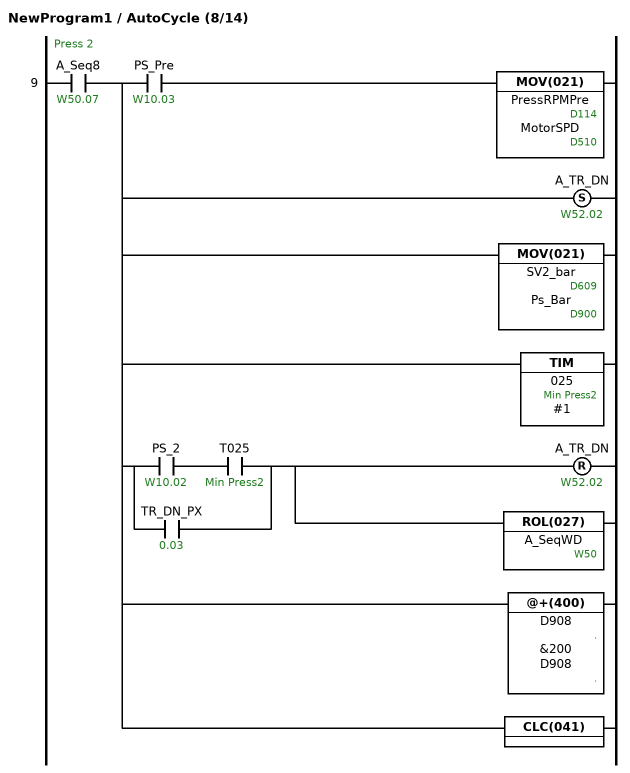
; [picture p24: NewProgram1 / AutoCycle, rungs 9-9]
; rung 9: Press 2
LD A_Seq8  ; W50.07
OUT TR0
AND PS_Pre  ; W10.03
MOV(021) PressRPMPre MotorSPD  ; D114, D510
LD TR0
SET A_TR_DN  ; W52.02
MOV(021) SV2_bar Ps_Bar  ; D609, D900
TIM 025 #1  ; Min Press2
LD PS_2  ; W10.02
AND T025  ; Min Press2
OR TR_DN_PX  ; 0.03
ANDLD
RSET A_TR_DN  ; W52.02
ROL(027) A_SeqWD  ; W50
LD TR0
@+(400) D908 &200 D908  ; .
CLC(041)

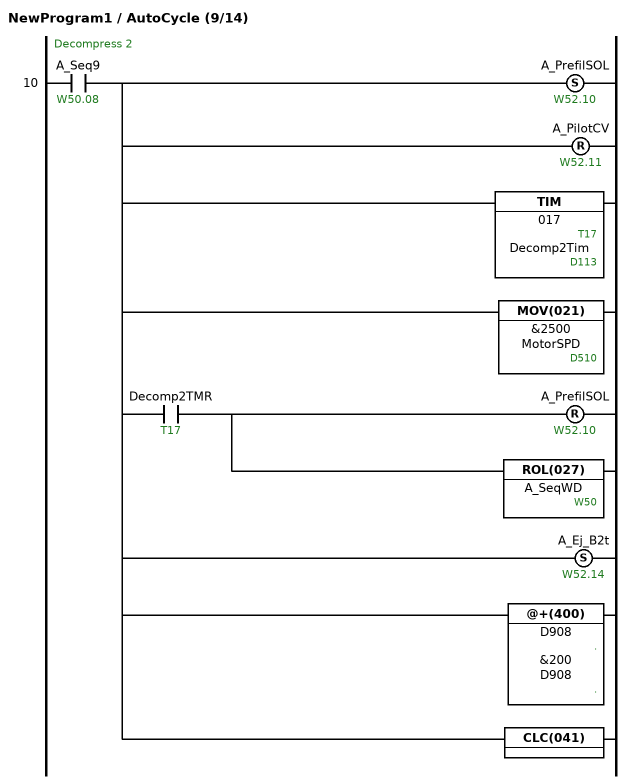
; rung 10: Decompress 2
LD A_Seq9  ; W50.08
OUT TR0
SET A_PrefilSOL  ; W52.10
RSET A_PilotCV  ; W52.11
TIM 017 Decomp2Tim  ; D113, T17
MOV(021) &2500 MotorSPD  ; D510
AND Decomp2TMR  ; T17
RSET A_PrefilSOL  ; W52.10
ROL(027) A_SeqWD  ; W50
LD TR0
SET A_Ej_B2t  ; W52.14
@+(400) D908 &200 D908  ; .
CLC(041)

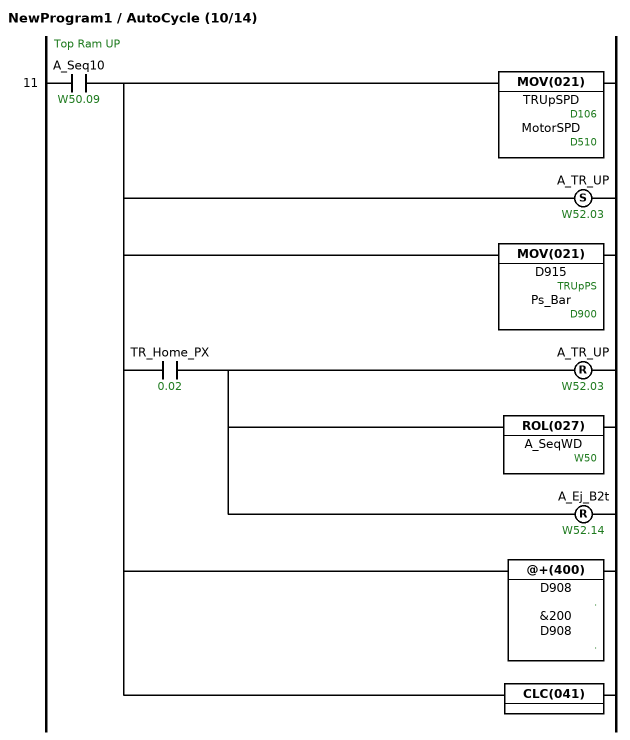
; rung 11: Top Ram UP
LD A_Seq10  ; W50.09
OUT TR0
MOV(021) TRUpSPD MotorSPD  ; D106, D510
SET A_TR_UP  ; W52.03
MOV(021) D915 Ps_Bar  ; TRUpPS, D900
AND TR_Home_PX  ; 0.02
RSET A_TR_UP  ; W52.03
ROL(027) A_SeqWD  ; W50
RSET A_Ej_B2t  ; W52.14
LD TR0
@+(400) D908 &200 D908  ; .
CLC(041)

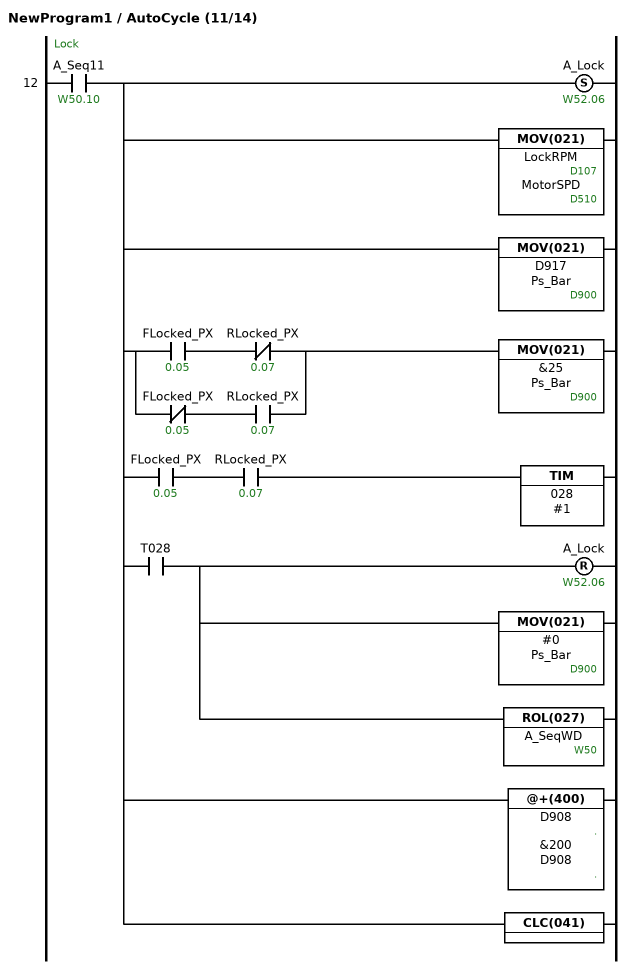
; rung 12: Lock
LD A_Seq11  ; W50.10
OUT TR0
SET A_Lock  ; W52.06
MOV(021) LockRPM MotorSPD  ; D107, D510
MOV(021) D917 Ps_Bar  ; D900
LD FLocked_PX  ; 0.05
ANDNOT RLocked_PX  ; 0.07
LDNOT FLocked_PX  ; 0.05
AND RLocked_PX  ; 0.07
ORLD
ANDLD
MOV(021) &25 Ps_Bar  ; D900
LD TR0
AND FLocked_PX  ; 0.05
AND RLocked_PX  ; 0.07
TIM 028 #1
LD TR0
AND T028
RSET A_Lock  ; W52.06
MOV(021) #0 Ps_Bar  ; D900
ROL(027) A_SeqWD  ; W50
LD TR0
@+(400) D908 &200 D908  ; .
CLC(041)

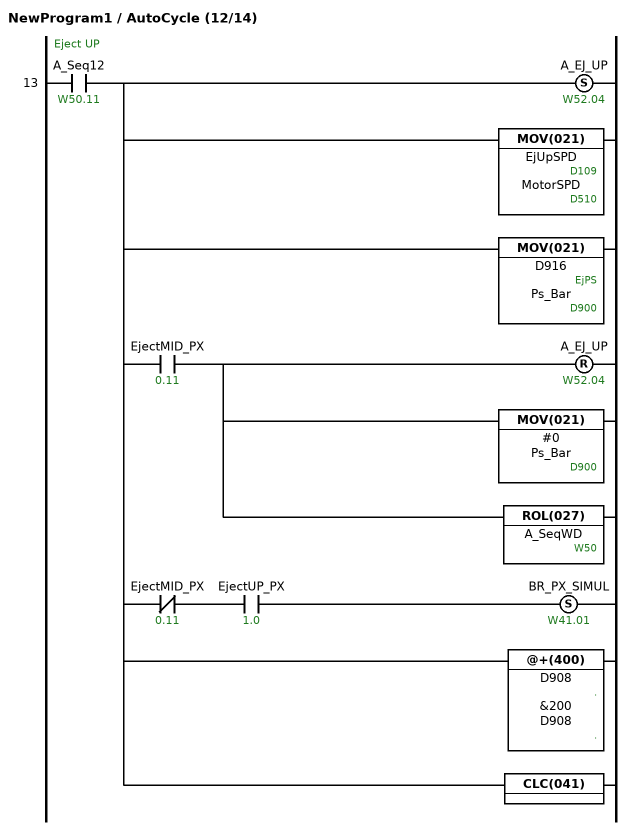
; rung 13: Eject UP
LD A_Seq12  ; W50.11
OUT TR0
SET A_EJ_UP  ; W52.04
MOV(021) EjUpSPD MotorSPD  ; D109, D510
MOV(021) D916 Ps_Bar  ; EjPS, D900
AND EjectMID_PX  ; 0.11
RSET A_EJ_UP  ; W52.04
MOV(021) #0 Ps_Bar  ; D900
ROL(027) A_SeqWD  ; W50
LD TR0
ANDNOT EjectMID_PX  ; 0.11
AND EjectUP_PX  ; 1.0
SET BR_PX_SIMUL  ; W41.01
LD TR0
@+(400) D908 &200 D908  ; .
CLC(041)

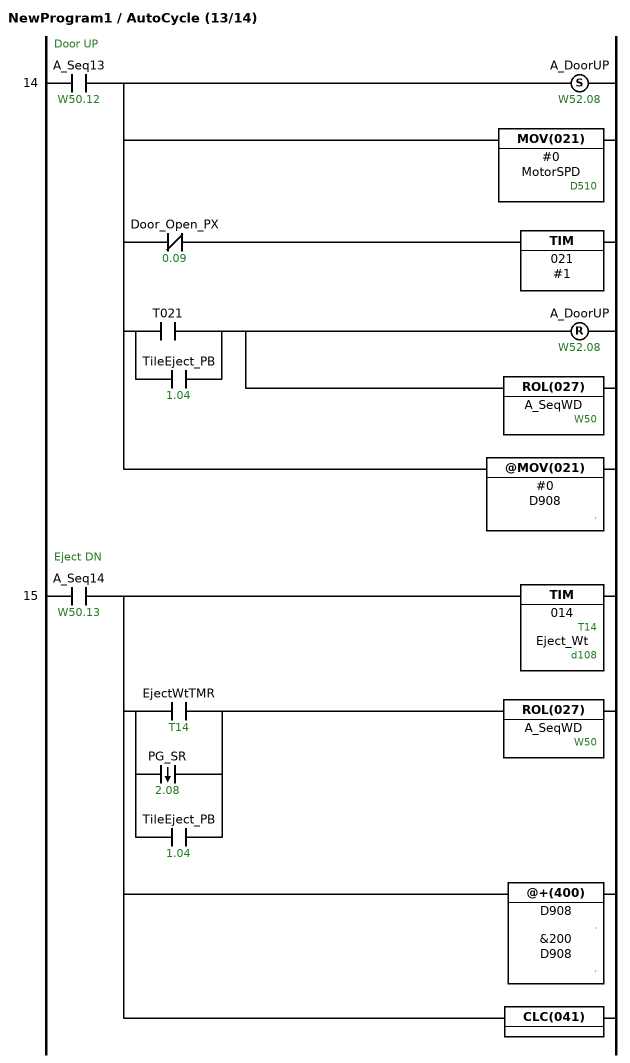
; rung 14: Door UP
LD A_Seq13  ; W50.12
OUT TR0
SET A_DoorUP  ; W52.08
MOV(021) #0 MotorSPD  ; D510
ANDNOT Door_Open_PX  ; 0.09
TIM 021 #1
LD TR0
LD T021
OR TileEject_PB  ; 1.04
ANDLD
RSET A_DoorUP  ; W52.08
ROL(027) A_SeqWD  ; W50
LD TR0
@MOV(021) #0 D908  ; .
; rung 15: Eject DN
LD A_Seq14  ; W50.13
OUT TR0
TIM 014 Eject_Wt  ; d108, T14
LD EjectWtTMR  ; T14
%OR PG_SR  ; 2.08
OR TileEject_PB  ; 1.04
ANDLD
ROL(027) A_SeqWD  ; W50
LD TR0
@+(400) D908 &200 D908  ; .
CLC(041)

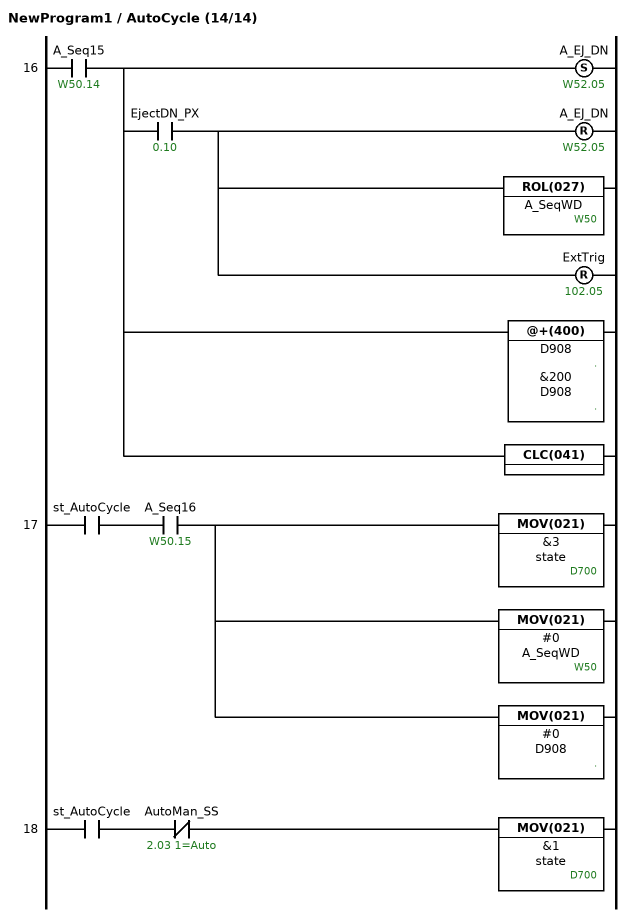
; rung 16
LD A_Seq15  ; W50.14
OUT TR0
SET A_EJ_DN  ; W52.05
AND EjectDN_PX  ; 0.10
RSET A_EJ_DN  ; W52.05
ROL(027) A_SeqWD  ; W50
RSET ExtTrig  ; 102.05
LD TR0
@+(400) D908 &200 D908  ; .
CLC(041)
; rung 17
LD st_AutoCycle
AND A_Seq16  ; W50.15
MOV(021) &3 state  ; D700
MOV(021) #0 A_SeqWD  ; W50
MOV(021) #0 D908  ; .
; rung 18
LD st_AutoCycle
ANDNOT AutoMan_SS  ; 2.03 1=Auto
MOV(021) &1 state  ; D700

### Section AutoReq

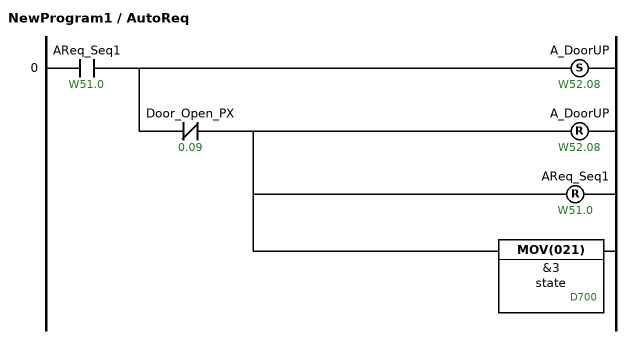
; rung 0
LD AReq_Seq1  ; W51.0
SET A_DoorUP  ; W52.08
ANDNOT Door_Open_PX  ; 0.09
RSET A_DoorUP  ; W52.08
RSET AReq_Seq1  ; W51.0
MOV(021) &3 state  ; D700

### Section TileEject

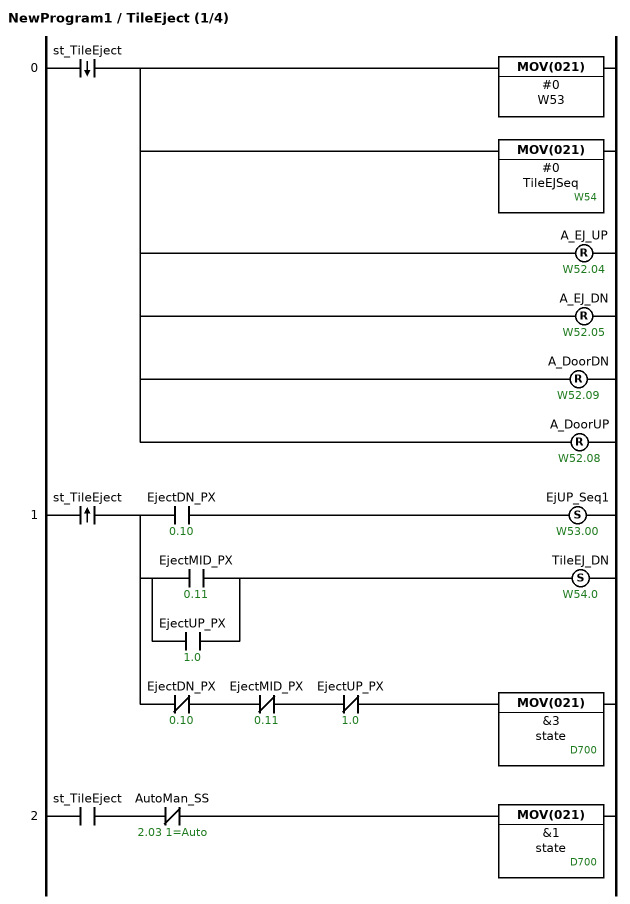
; rung 0
%LD st_TileEject
MOV(021) #0 W53
MOV(021) #0 TileEJSeq  ; W54
RSET A_EJ_UP  ; W52.04
RSET A_EJ_DN  ; W52.05
RSET A_DoorDN  ; W52.09
RSET A_DoorUP  ; W52.08
; rung 1
@LD st_TileEject
OUT TR0
AND EjectDN_PX  ; 0.10
SET EjUP_Seq1  ; W53.00
LD TR0
LD EjectMID_PX  ; 0.11
OR EjectUP_PX  ; 1.0
ANDLD
SET TileEJ_DN  ; W54.0
LD TR0
ANDNOT EjectDN_PX  ; 0.10
ANDNOT EjectMID_PX  ; 0.11
ANDNOT EjectUP_PX  ; 1.0
MOV(021) &3 state  ; D700
; rung 2
LD st_TileEject
ANDNOT AutoMan_SS  ; 2.03 1=Auto
MOV(021) &1 state  ; D700

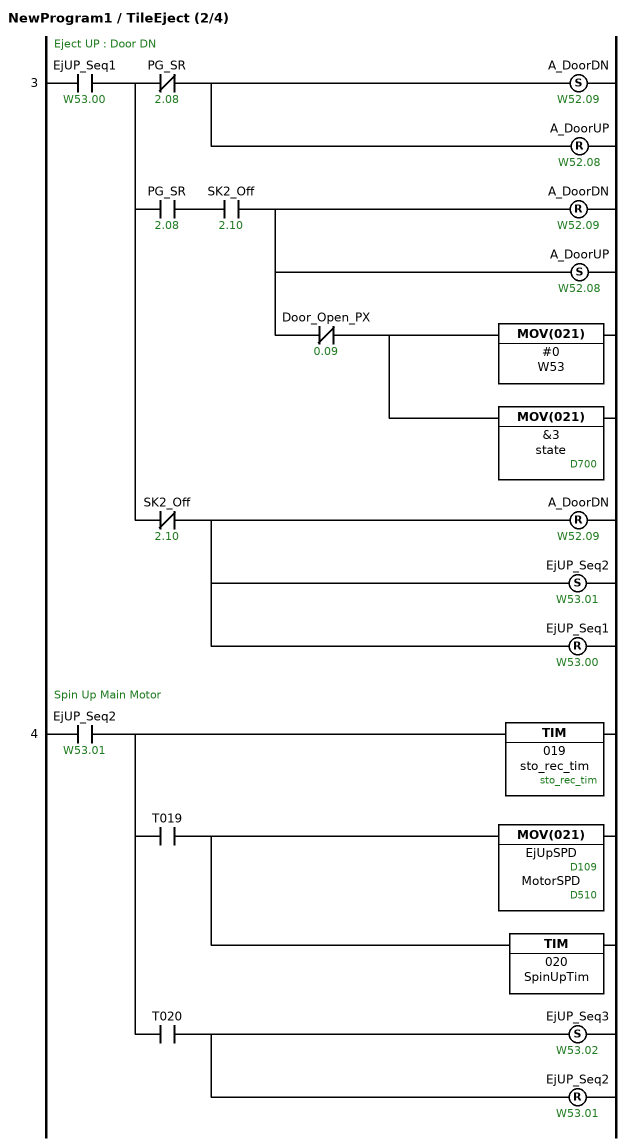
; rung 3: Eject UP : Door DN
LD EjUP_Seq1  ; W53.00
OUT TR0
ANDNOT PG_SR  ; 2.08
SET A_DoorDN  ; W52.09
RSET A_DoorUP  ; W52.08
LD TR0
AND PG_SR  ; 2.08
AND SK2_Off  ; 2.10
RSET A_DoorDN  ; W52.09
SET A_DoorUP  ; W52.08
ANDNOT Door_Open_PX  ; 0.09
MOV(021) #0 W53
MOV(021) &3 state  ; D700
LD TR0
ANDNOT SK2_Off  ; 2.10
RSET A_DoorDN  ; W52.09
SET EjUP_Seq2  ; W53.01
RSET EjUP_Seq1  ; W53.00
; rung 4: Spin Up Main Motor
LD EjUP_Seq2  ; W53.01
OUT TR0
TIM 019 sto_rec_tim  ; sto_rec_tim
AND T019
MOV(021) EjUpSPD MotorSPD  ; D109, D510
TIM 020 SpinUpTim
LD TR0
AND T020
SET EjUP_Seq3  ; W53.02
RSET EjUP_Seq2  ; W53.01

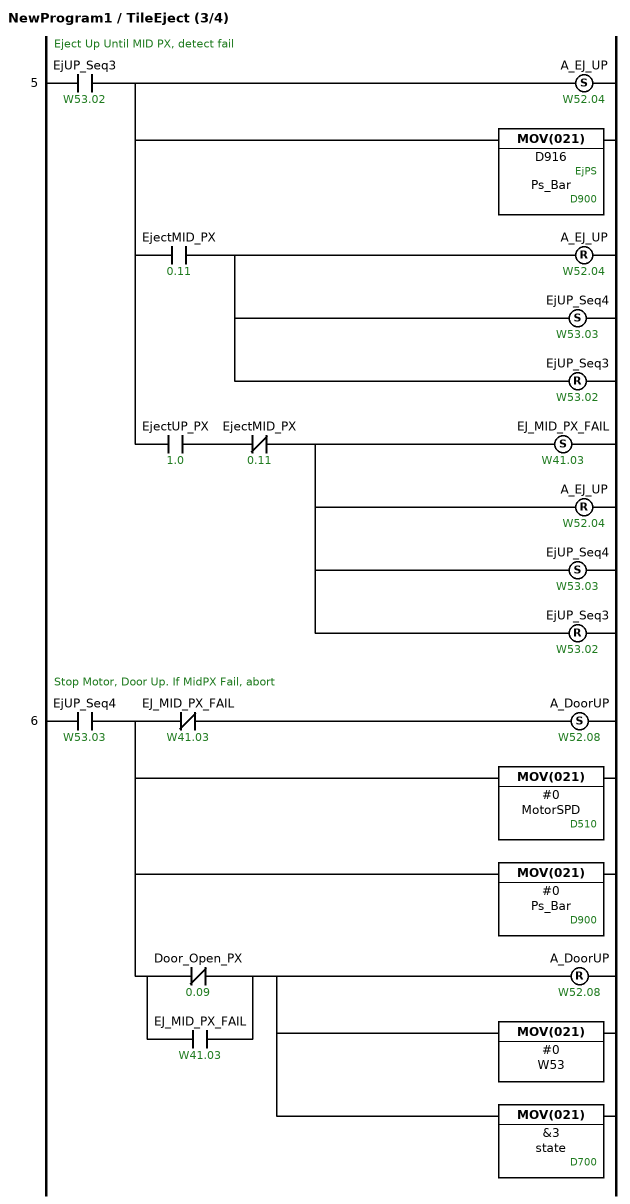
; rung 5: Eject Up Until MID PX, detect fail
LD EjUP_Seq3  ; W53.02
OUT TR0
SET A_EJ_UP  ; W52.04
MOV(021) D916 Ps_Bar  ; EjPS, D900
AND EjectMID_PX  ; 0.11
RSET A_EJ_UP  ; W52.04
SET EjUP_Seq4  ; W53.03
RSET EjUP_Seq3  ; W53.02
LD TR0
AND EjectUP_PX  ; 1.0
ANDNOT EjectMID_PX  ; 0.11
SET EJ_MID_PX_FAIL  ; W41.03
RSET A_EJ_UP  ; W52.04
SET EjUP_Seq4  ; W53.03
RSET EjUP_Seq3  ; W53.02
; rung 6: Stop Motor, Door Up. If MidPX Fail, abort
LD EjUP_Seq4  ; W53.03
OUT TR0
ANDNOT EJ_MID_PX_FAIL  ; W41.03
SET A_DoorUP  ; W52.08
LD TR0
MOV(021) #0 MotorSPD  ; D510
MOV(021) #0 Ps_Bar  ; D900
LDNOT Door_Open_PX  ; 0.09
OR EJ_MID_PX_FAIL  ; W41.03
ANDLD
RSET A_DoorUP  ; W52.08
MOV(021) #0 W53
MOV(021) &3 state  ; D700

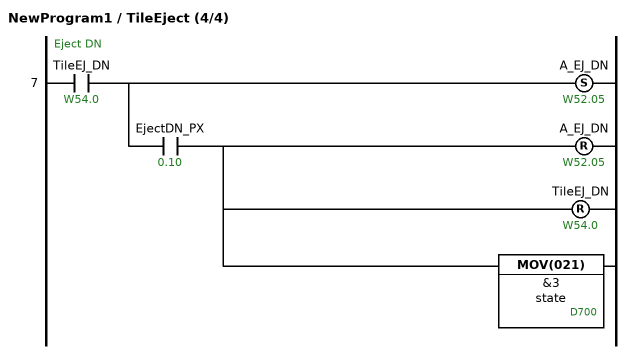
; rung 7: Eject DN
LD TileEJ_DN  ; W54.0
SET A_EJ_DN  ; W52.05
AND EjectDN_PX  ; 0.10
RSET A_EJ_DN  ; W52.05
RSET TileEJ_DN  ; W54.0
MOV(021) &3 state  ; D700

### Section MainMotorCtrl
; rung 0: 14.57 -> 3000, 14.59-> 3000

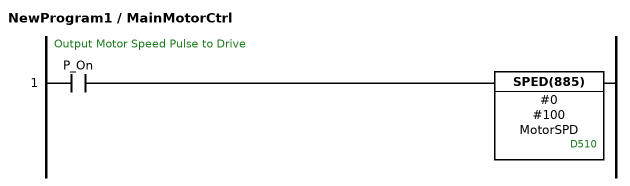
; rung 1: Output Motor Speed Pulse to Drive
LD P_On
SPED(885) #0 #100 MotorSPD  ; D510

### Section Outputs

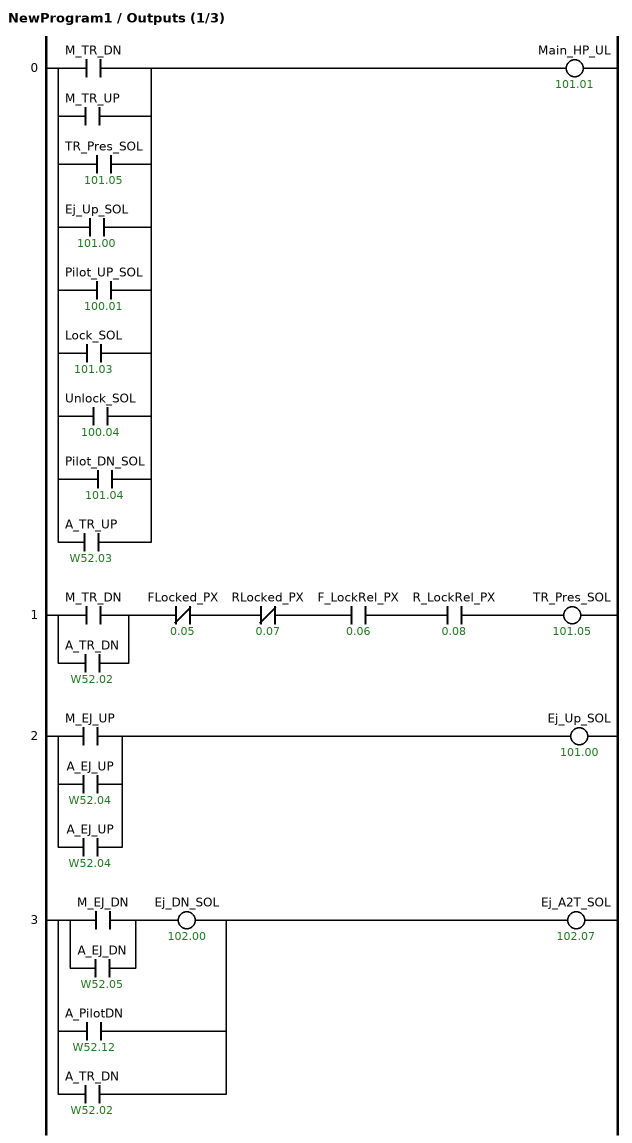
; rung 0
LD M_TR_DN
OR M_TR_UP
OR TR_Pres_SOL  ; 101.05
OR Ej_Up_SOL  ; 101.00
OR Pilot_UP_SOL  ; 100.01
OR Lock_SOL  ; 101.03
OR Unlock_SOL  ; 100.04
OR Pilot_DN_SOL  ; 101.04
OR A_TR_UP  ; W52.03
OUT Main_HP_UL  ; 101.01
; rung 1
LD M_TR_DN
OR A_TR_DN  ; W52.02
ANDNOT FLocked_PX  ; 0.05
ANDNOT RLocked_PX  ; 0.07
AND F_LockRel_PX  ; 0.06
AND R_LockRel_PX  ; 0.08
OUT TR_Pres_SOL  ; 101.05
; rung 2
LD M_EJ_UP
OR A_EJ_UP  ; W52.04
OR A_EJ_UP  ; W52.04
OUT Ej_Up_SOL  ; 101.00
; rung 3
LD M_EJ_DN
OR A_EJ_DN  ; W52.05
OUT Ej_DN_SOL  ; 102.00
LD A_PilotDN  ; W52.12
OR A_TR_DN  ; W52.02
ORLD
OUT Ej_A2T_SOL  ; 102.07

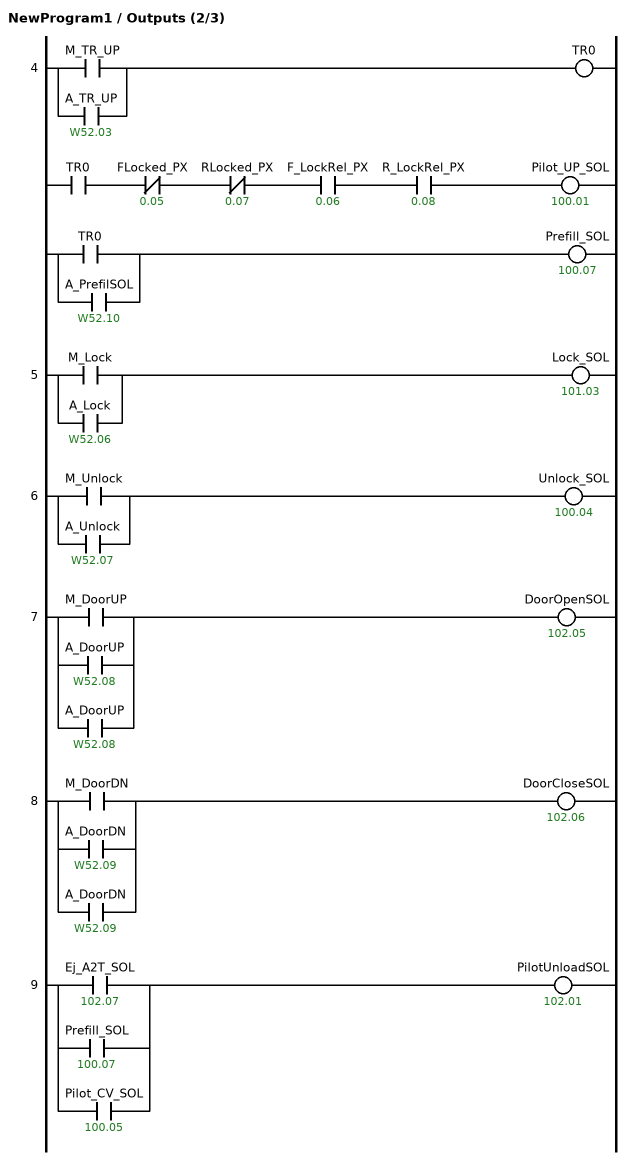
; rung 4
LD M_TR_UP
OR A_TR_UP  ; W52.03
OUT TR0
ANDNOT FLocked_PX  ; 0.05
ANDNOT RLocked_PX  ; 0.07
AND F_LockRel_PX  ; 0.06
AND R_LockRel_PX  ; 0.08
OUT Pilot_UP_SOL  ; 100.01
LD TR0
OR A_PrefilSOL  ; W52.10
OUT Prefill_SOL  ; 100.07
; rung 5
LD M_Lock
OR A_Lock  ; W52.06
OUT Lock_SOL  ; 101.03
; rung 6
LD M_Unlock
OR A_Unlock  ; W52.07
OUT Unlock_SOL  ; 100.04
; rung 7
LD M_DoorUP
OR A_DoorUP  ; W52.08
OR A_DoorUP  ; W52.08
OUT DoorOpenSOL  ; 102.05
; rung 8
LD M_DoorDN
OR A_DoorDN  ; W52.09
OR A_DoorDN  ; W52.09
OUT DoorCloseSOL  ; 102.06
; rung 9
LD Ej_A2T_SOL  ; 102.07
OR Prefill_SOL  ; 100.07
OR Pilot_CV_SOL  ; 100.05
OUT PilotUnloadSOL  ; 102.01

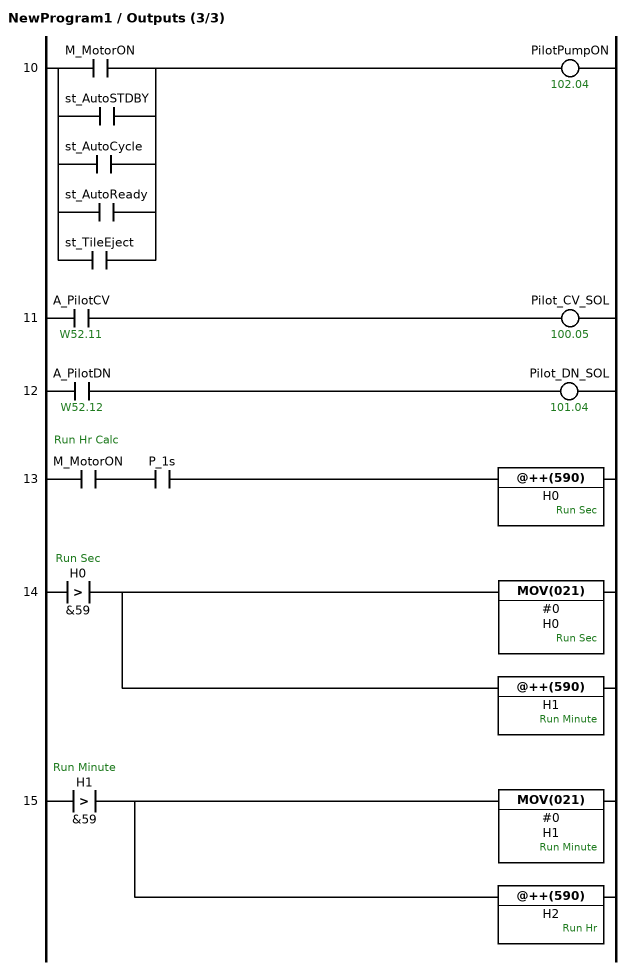
; rung 10
LD M_MotorON
OR st_AutoSTDBY
OR st_AutoCycle
OR st_AutoReady
OR st_TileEject
OUT PilotPumpON  ; 102.04
; rung 11
LD A_PilotCV  ; W52.11
OUT Pilot_CV_SOL  ; 100.05
; rung 12
LD A_PilotDN  ; W52.12
OUT Pilot_DN_SOL  ; 101.04
; rung 13: Run Hr Calc
LD M_MotorON
AND P_1s
@++(590) H0  ; Run Sec
; rung 14
LD>(320) H0 &59  ; Run Sec
MOV(021) #0 H0  ; Run Sec
@++(590) H1  ; Run Minute
; rung 15
LD>(320) H1 &59  ; Run Minute
MOV(021) #0 H1  ; Run Minute
@++(590) H2  ; Run Hr

### Section Profile

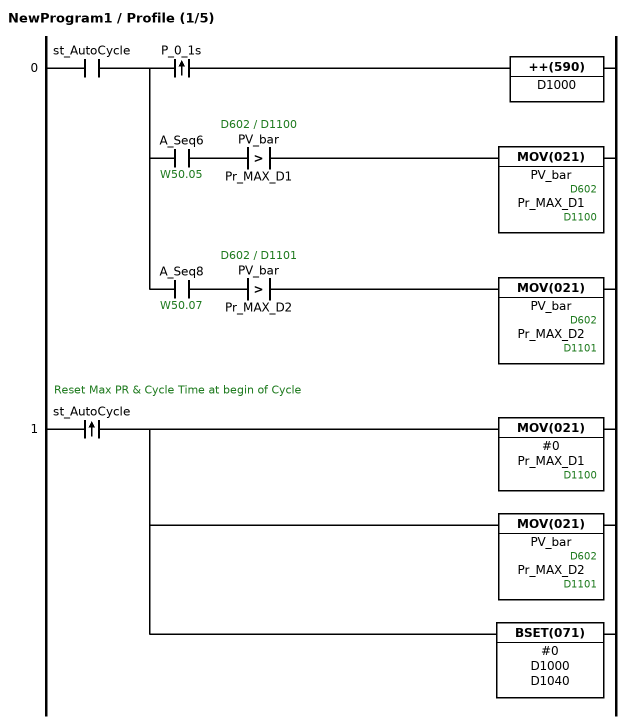
; rung 0
LD st_AutoCycle
OUT TR0
@AND P_0_1s
++(590) D1000
LD TR0
AND A_Seq6  ; W50.05
AND>(320) PV_bar Pr_MAX_D1  ; D602, D1100
MOV(021) PV_bar Pr_MAX_D1  ; D602, D1100
LD TR0
AND A_Seq8  ; W50.07
AND>(320) PV_bar Pr_MAX_D2  ; D602, D1101
MOV(021) PV_bar Pr_MAX_D2  ; D602, D1101
; rung 1: Reset Max PR & Cycle Time at begin of Cycle
@LD st_AutoCycle
MOV(021) #0 Pr_MAX_D1  ; D1100
MOV(021) PV_bar Pr_MAX_D2  ; D602, D1101
BSET(071) #0 D1000 D1040

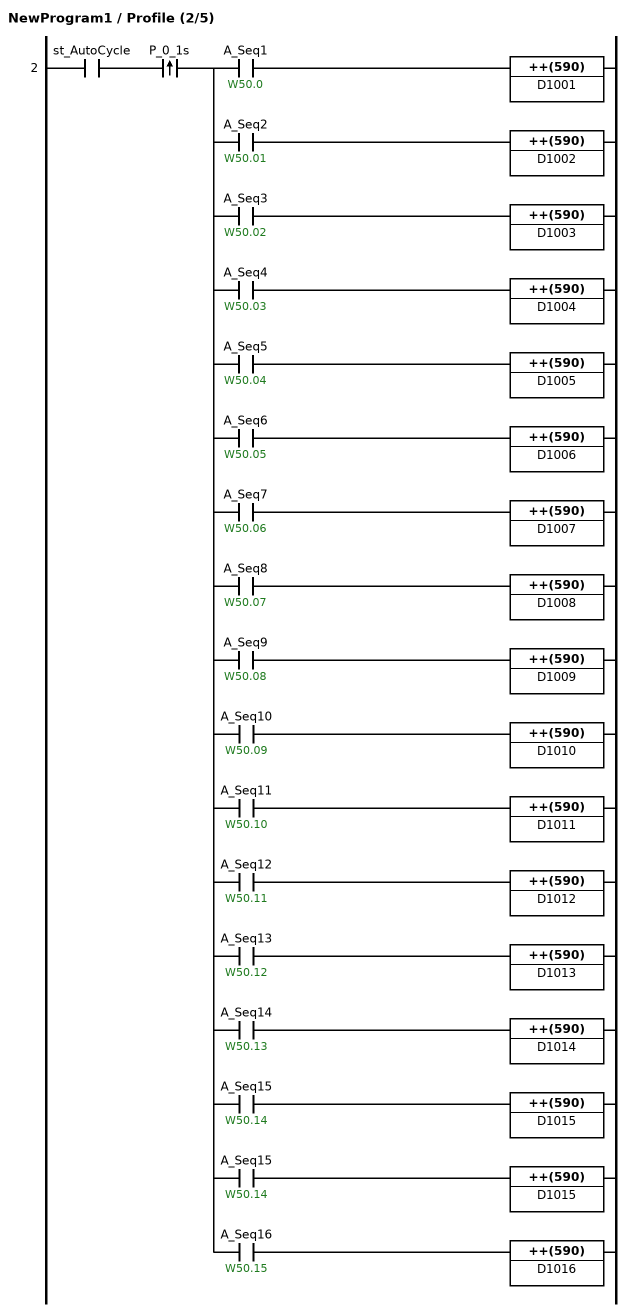
; rung 2
LD st_AutoCycle
@AND P_0_1s
OUT TR0
AND A_Seq1  ; W50.0
++(590) D1001
LD TR0
AND A_Seq2  ; W50.01
++(590) D1002
LD TR0
AND A_Seq3  ; W50.02
++(590) D1003
LD TR0
AND A_Seq4  ; W50.03
++(590) D1004
LD TR0
AND A_Seq5  ; W50.04
++(590) D1005
LD TR0
AND A_Seq6  ; W50.05
++(590) D1006
LD TR0
AND A_Seq7  ; W50.06
++(590) D1007
LD TR0
AND A_Seq8  ; W50.07
++(590) D1008
LD TR0
AND A_Seq9  ; W50.08
++(590) D1009
LD TR0
AND A_Seq10  ; W50.09
++(590) D1010
LD TR0
AND A_Seq11  ; W50.10
++(590) D1011
LD TR0
AND A_Seq12  ; W50.11
++(590) D1012
LD TR0
AND A_Seq13  ; W50.12
++(590) D1013
LD TR0
AND A_Seq14  ; W50.13
++(590) D1014
LD TR0
AND A_Seq15  ; W50.14
++(590) D1015
LD TR0
AND A_Seq15  ; W50.14
++(590) D1015
LD TR0
AND A_Seq16  ; W50.15
++(590) D1016

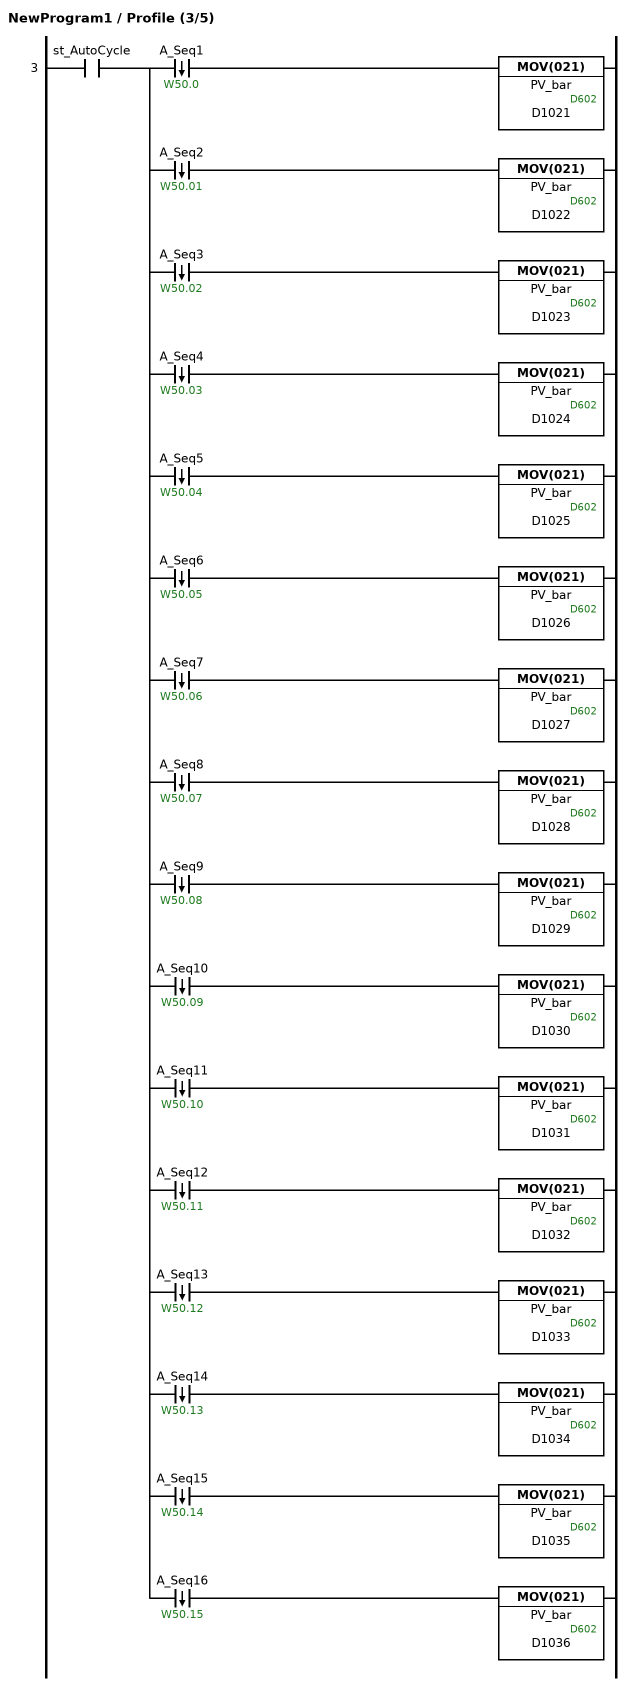
; rung 3
LD st_AutoCycle
OUT TR0
%AND A_Seq1  ; W50.0
MOV(021) PV_bar D1021  ; D602
LD TR0
%AND A_Seq2  ; W50.01
MOV(021) PV_bar D1022  ; D602
LD TR0
%AND A_Seq3  ; W50.02
MOV(021) PV_bar D1023  ; D602
LD TR0
%AND A_Seq4  ; W50.03
MOV(021) PV_bar D1024  ; D602
LD TR0
%AND A_Seq5  ; W50.04
MOV(021) PV_bar D1025  ; D602
LD TR0
%AND A_Seq6  ; W50.05
MOV(021) PV_bar D1026  ; D602
LD TR0
%AND A_Seq7  ; W50.06
MOV(021) PV_bar D1027  ; D602
LD TR0
%AND A_Seq8  ; W50.07
MOV(021) PV_bar D1028  ; D602
LD TR0
%AND A_Seq9  ; W50.08
MOV(021) PV_bar D1029  ; D602
LD TR0
%AND A_Seq10  ; W50.09
MOV(021) PV_bar D1030  ; D602
LD TR0
%AND A_Seq11  ; W50.10
MOV(021) PV_bar D1031  ; D602
LD TR0
%AND A_Seq12  ; W50.11
MOV(021) PV_bar D1032  ; D602
LD TR0
%AND A_Seq13  ; W50.12
MOV(021) PV_bar D1033  ; D602
LD TR0
%AND A_Seq14  ; W50.13
MOV(021) PV_bar D1034  ; D602
LD TR0
%AND A_Seq15  ; W50.14
MOV(021) PV_bar D1035  ; D602
LD TR0
%AND A_Seq16  ; W50.15
MOV(021) PV_bar D1036  ; D602

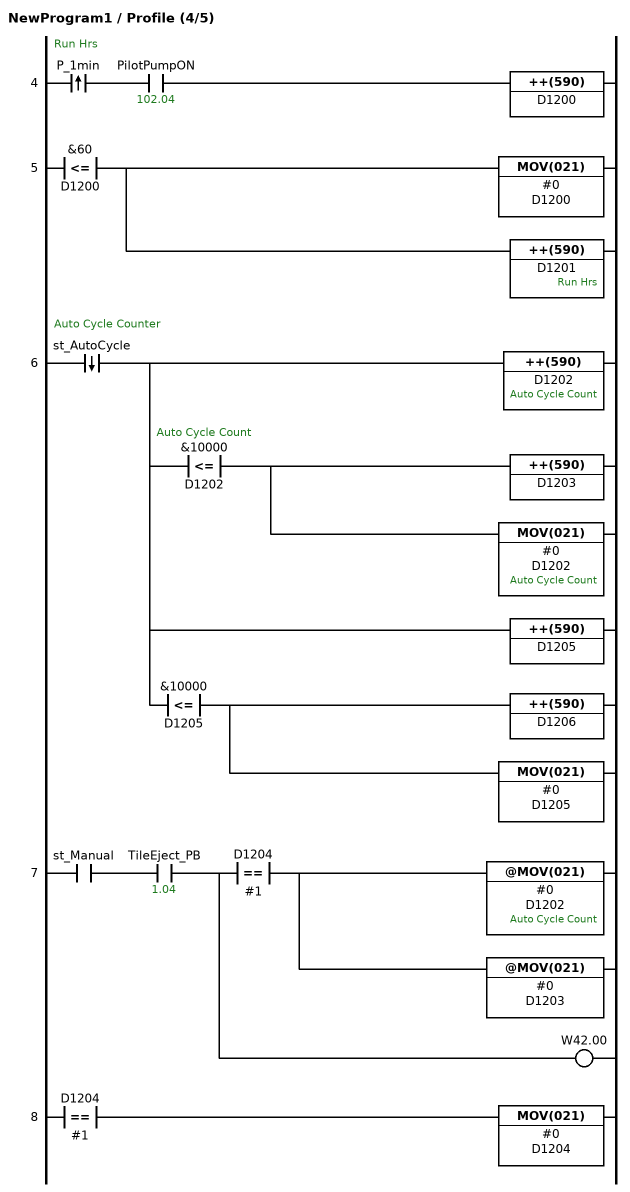
; rung 4: Run Hrs
@LD P_1min
AND PilotPumpON  ; 102.04
++(590) D1200
; rung 5
LD<=(315) &60 D1200
MOV(021) #0 D1200
++(590) D1201  ; Run Hrs
; rung 6: Auto Cycle Counter
%LD st_AutoCycle
OUT TR0
++(590) D1202  ; Auto Cycle Count
AND<=(315) &10000 D1202  ; Auto Cycle Count
++(590) D1203
MOV(021) #0 D1202  ; Auto Cycle Count
LD TR0
++(590) D1205
AND<=(315) &10000 D1205
++(590) D1206
MOV(021) #0 D1205
; rung 7
LD st_Manual
AND TileEject_PB  ; 1.04
OUT TR0
AND=(300) D1204 #1
@MOV(021) #0 D1202  ; Auto Cycle Count
@MOV(021) #0 D1203
LD TR0
OUT W42.00
; rung 8
LD=(300) D1204 #1
MOV(021) #0 D1204

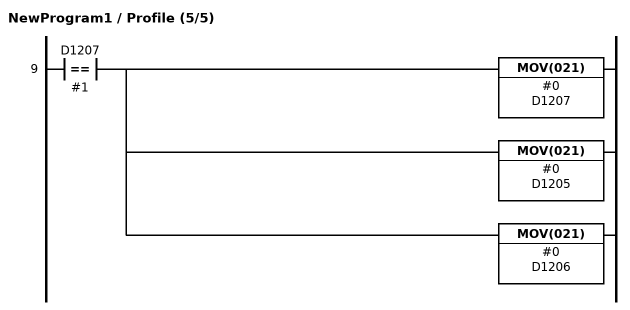
; rung 9
LD=(300) D1207 #1
MOV(021) #0 D1207
MOV(021) #0 D1205
MOV(021) #0 D1206

### Section HMI

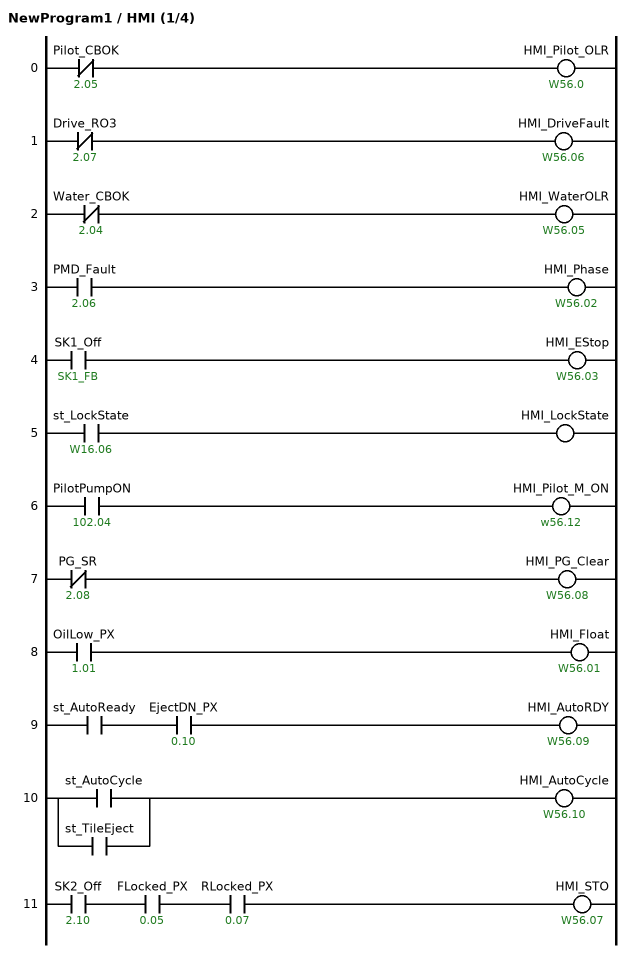
; rung 0
LDNOT Pilot_CBOK  ; 2.05
OUT HMI_Pilot_OLR  ; W56.0
; rung 1
LDNOT Drive_RO3  ; 2.07
OUT HMI_DriveFault  ; W56.06
; rung 2
LDNOT Water_CBOK  ; 2.04
OUT HMI_WaterOLR  ; W56.05
; rung 3
LD PMD_Fault  ; 2.06
OUT HMI_Phase  ; W56.02
; rung 4
LD SK1_Off  ; SK1_FB
OUT HMI_EStop  ; W56.03
; rung 5
LD st_LockState  ; W16.06
OUT HMI_LockState
; rung 6
LD PilotPumpON  ; 102.04
OUT HMI_Pilot_M_ON  ; w56.12
; rung 7
LDNOT PG_SR  ; 2.08
OUT HMI_PG_Clear  ; W56.08
; rung 8
LD OilLow_PX  ; 1.01
OUT HMI_Float  ; W56.01
; rung 9
LD st_AutoReady
AND EjectDN_PX  ; 0.10
OUT HMI_AutoRDY  ; W56.09
; rung 10
LD st_AutoCycle
OR st_TileEject
OUT HMI_AutoCycle  ; W56.10
; rung 11
LD SK2_Off  ; 2.10
AND FLocked_PX  ; 0.05
AND RLocked_PX  ; 0.07
OUT HMI_STO  ; W56.07

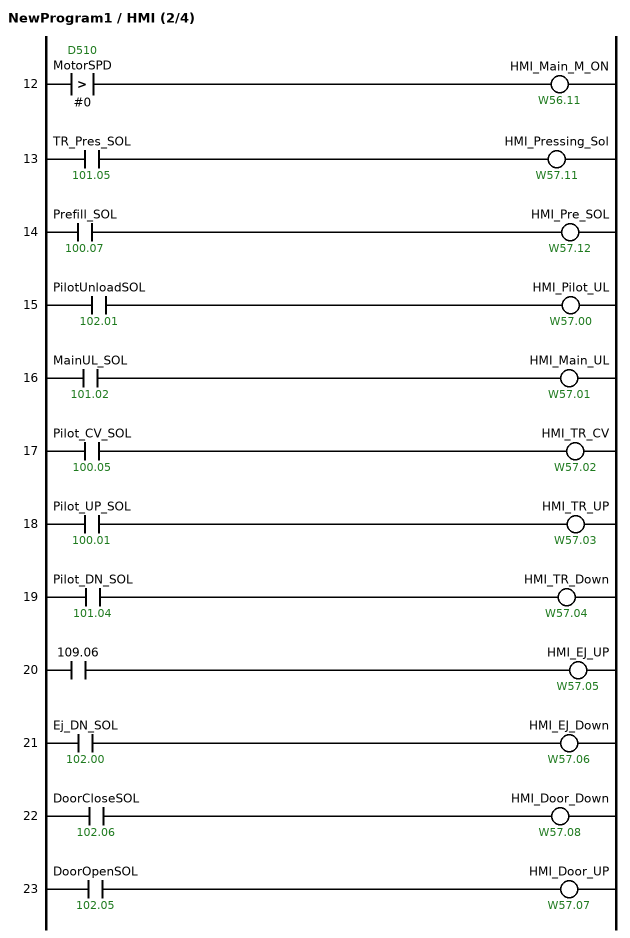
; rung 12
LD>(320) MotorSPD #0  ; D510
OUT HMI_Main_M_ON  ; W56.11
; rung 13
LD TR_Pres_SOL  ; 101.05
OUT HMI_Pressing_Sol  ; W57.11
; rung 14
LD Prefill_SOL  ; 100.07
OUT HMI_Pre_SOL  ; W57.12
; rung 15
LD PilotUnloadSOL  ; 102.01
OUT HMI_Pilot_UL  ; W57.00
; rung 16
LD MainUL_SOL  ; 101.02
OUT HMI_Main_UL  ; W57.01
; rung 17
LD Pilot_CV_SOL  ; 100.05
OUT HMI_TR_CV  ; W57.02
; rung 18
LD Pilot_UP_SOL  ; 100.01
OUT HMI_TR_UP  ; W57.03
; rung 19
LD Pilot_DN_SOL  ; 101.04
OUT HMI_TR_Down  ; W57.04
; rung 20
LD 109.06
OUT HMI_EJ_UP  ; W57.05
; rung 21
LD Ej_DN_SOL  ; 102.00
OUT HMI_EJ_Down  ; W57.06
; rung 22
LD DoorCloseSOL  ; 102.06
OUT HMI_Door_Down  ; W57.08
; rung 23
LD DoorOpenSOL  ; 102.05
OUT HMI_Door_UP  ; W57.07

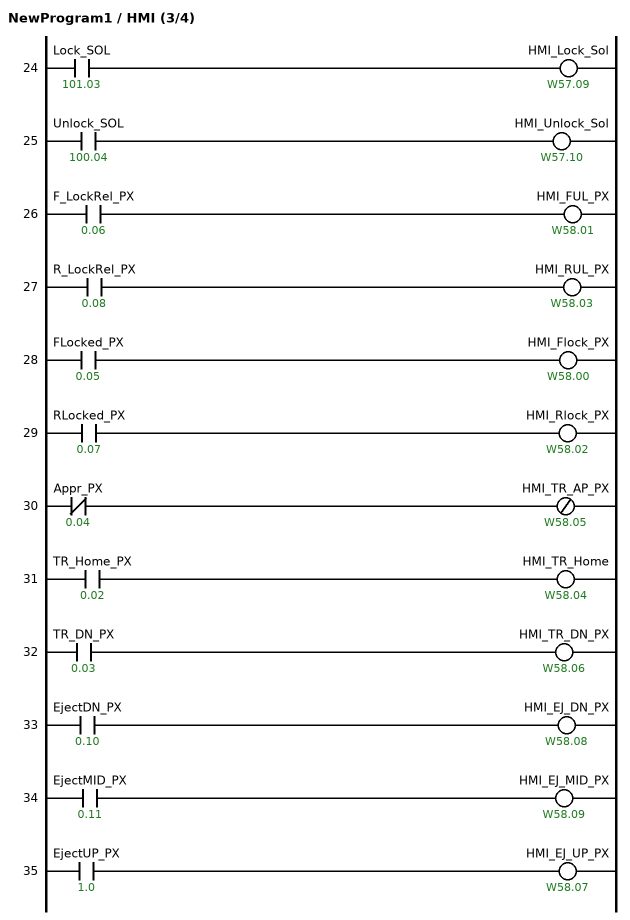
; rung 24
LD Lock_SOL  ; 101.03
OUT HMI_Lock_Sol  ; W57.09
; rung 25
LD Unlock_SOL  ; 100.04
OUT HMI_Unlock_Sol  ; W57.10
; rung 26
LD F_LockRel_PX  ; 0.06
OUT HMI_FUL_PX  ; W58.01
; rung 27
LD R_LockRel_PX  ; 0.08
OUT HMI_RUL_PX  ; W58.03
; rung 28
LD FLocked_PX  ; 0.05
OUT HMI_Flock_PX  ; W58.00
; rung 29
LD RLocked_PX  ; 0.07
OUT HMI_Rlock_PX  ; W58.02
; rung 30
LDNOT Appr_PX  ; 0.04
OUTNOT HMI_TR_AP_PX  ; W58.05
; rung 31
LD TR_Home_PX  ; 0.02
OUT HMI_TR_Home  ; W58.04
; rung 32
LD TR_DN_PX  ; 0.03
OUT HMI_TR_DN_PX  ; W58.06
; rung 33
LD EjectDN_PX  ; 0.10
OUT HMI_EJ_DN_PX  ; W58.08
; rung 34
LD EjectMID_PX  ; 0.11
OUT HMI_EJ_MID_PX  ; W58.09
; rung 35
LD EjectUP_PX  ; 1.0
OUT HMI_EJ_UP_PX  ; W58.07

